(* IEC 61131-3 sources: Bachelor/LARS redcrane-simulation/plc_export/FB_InverceKinematicsVaribleTelescope (part 2) *)

                (* clear; clc; *)
                (* expc3 = [1; 2; 3]; *)
                (* [omghat, theta] = AxisAng3(expc3)   *)

                (* Output: *)
                (* omghat = *)
                (* 0.2673 *)
                (* 0.5345 *)
                (* 0.8018 *)
                (* theta = *)
                (* 3.7417 *)
                (* 'AxisAng3:20' theta = norm(expc3); *)
                (* 'AxisAng3:21' omghat = expc3 / theta; *)
                (* 'MatrixExp6:27' omgmat = se3mat(1: 3, 1: 3) / theta; *)
                FOR i_0 := 0 TO 2 DO
                    omgmat_tmp := DWORD_TO_DINT(SHL(DINT_TO_DWORD(i_0), 2));
                    omgmat[3 * i_0] := se3mat[omgmat_tmp] / c_theta;
                    omgmat[(3 * i_0) + 1] := se3mat[omgmat_tmp + 1] / c_theta;
                    omgmat[(3 * i_0) + 2] := se3mat[omgmat_tmp + 2] / c_theta;
                END_FOR;
                (* 'MatrixExp6:28' T = [MatrixExp3(se3mat(1: 3, 1: 3)), ... *)
                (* 'MatrixExp6:29'          (eye(3) * theta + (1 - cos(theta)) * omgmat ... *)
                (* 'MatrixExp6:30'           + (theta - sin(theta)) * omgmat * omgmat) ... *)
                (* 'MatrixExp6:31'             * se3mat(1: 3, 4) / theta; *)
                (* 'MatrixExp6:32'          0, 0, 0, 1]; *)
                thetalist0_0 := 1.0 - COS(c_theta);
                g_a := c_theta - SIN(c_theta);
                (* *** CHAPTER 3: RIGID-BODY MOTIONS *** *)
                (* Takes a 3x3 so(3) representation of exponential coordinates. *)
                (* Returns R in SO(3) that is achieved by rotating about omghat by theta  *)
                (* from an initial orientation R = I. *)
                (* Example Input: *)

                (* clear; clc; *)
                (* so3mat = [[0, -3, 2]; [3, 0, -1]; [-2, 1, 0]]; *)
                (* R = MatrixExp3(so3mat)   *)

                (* Output: *)
                (* R = *)
                (* -0.6949    0.7135    0.0893 *)
                (* -0.1920   -0.3038    0.9332 *)
                (* 0.6930    0.6313    0.3481 *)
                (* 'MatrixExp3:18' omgtheta = so3ToVec(so3mat); *)
                (* *** CHAPTER 3: RIGID-BODY MOTIONS *** *)
                (* Takes a 3x3 skew-symmetric matrix (an element of so(3)). *)
                (* Returns the corresponding 3-vector (angular velocity). *)
                (* Example Input:  *)

                (* clear; clc; *)
                (* so3mat = [[0, -3, 2]; [3, 0, -1]; [-2, 1, 0]]; *)
                (* omg = so3ToVec(so3mat)   *)

                (* Output: *)
                (* omg = *)
                (* 1 *)
                (* 2 *)
                (* 3 *)
                (* 'so3ToVec:17' omg = [so3mat(3, 2); so3mat(1, 3); so3mat(2, 1)]; *)
                qs4[0] := V[0];
                qs4[1] := V[1];
                qs4[2] := V[2];
                (* 'MatrixExp3:19' if NearZero(norm(omgtheta)) *)
                (* *** BASIC HELPER FUNCTIONS *** *)
                (* Takes a scalar. *)
                (* Checks if the scalar is small enough to be neglected. *)
                (* Example Input: *)

                (* clear; clc; *)
                (* near = -1e-7; *)
                (* judge = NearZero(near) *)

                (* Output: *)
                (* judge = *)
                (* 1 *)
                (* 'NearZero:15' judge = norm(near) < 1e-6; *)
                i_theta := norm(x := qs4);
                IF ABS(i_theta) < 1.0E-6 THEN
                    (* 'MatrixExp3:20' R = eye(3); *)
                    i0_eye();
                    b_R := i0_eye.I;
                ELSE
                    (* 'MatrixExp3:21' else *)
                    (* 'MatrixExp3:22' [omghat, theta] = AxisAng3(omgtheta); *)
                    (* *** CHAPTER 3: RIGID-BODY MOTIONS *** *)
                    (* Takes A 3-vector of exponential coordinates for rotation. *)
                    (* Returns the unit rotation axis omghat and the corresponding rotation  *)
                    (* angle theta. *)
                    (* Example Input: *)

                    (* clear; clc; *)
                    (* expc3 = [1; 2; 3]; *)
                    (* [omghat, theta] = AxisAng3(expc3)   *)

                    (* Output: *)
                    (* omghat = *)
                    (* 0.2673 *)
                    (* 0.5345 *)
                    (* 0.8018 *)
                    (* theta = *)
                    (* 3.7417 *)
                    (* 'AxisAng3:20' theta = norm(expc3); *)
                    (* 'AxisAng3:21' omghat = expc3 / theta; *)
                    (* 'MatrixExp3:23' omgmat = so3mat / theta; *)
                    FOR i_0 := 0 TO 2 DO
                        omgmat_tmp := DWORD_TO_DINT(SHL(DINT_TO_DWORD(i_0), 2));
                        b_omgmat[3 * i_0] := se3mat[omgmat_tmp] / i_theta;
                        b_omgmat[(3 * i_0) + 1] := se3mat[omgmat_tmp + 1] / i_theta;
                        b_omgmat[(3 * i_0) + 2] := se3mat[omgmat_tmp + 2] / i_theta;
                    END_FOR;
                    (* 'MatrixExp3:24' R = eye(3) + sin(theta) * omgmat + (1 - cos(theta)) * omgmat * omgmat; *)
                    l_a := SIN(i_theta);
                    x_tmp := COS(i_theta);
                    i0_eye();
                    tmp := i0_eye.I;
                    FOR i_0 := 0 TO 2 DO
                        FOR omgmat_tmp := 0 TO 2 DO
                            R_tmp := (3 * omgmat_tmp) + i_0;
                            b_R[R_tmp] := (((((1.0 - x_tmp) * b_omgmat[i_0 + 3]) * b_omgmat[(3 * omgmat_tmp) + 1]) + (((1.0 - x_tmp) * b_omgmat[i_0]) * b_omgmat[3 * omgmat_tmp])) + ((b_omgmat[i_0 + 6] * (1.0 - x_tmp)) * b_omgmat[(3 * omgmat_tmp) + 2])) + ((b_omgmat[R_tmp] * l_a) + tmp[R_tmp]);
                        END_FOR;
                    END_FOR;
                END_IF;
                FOR i_0 := 0 TO 2 DO
                    x_tmp := 0.0;
                    FOR omgmat_tmp := 0 TO 2 DO
                        R_tmp := (3 * omgmat_tmp) + i_0;
                        x_tmp := ((((((omgmat[i_0 + 3] * g_a) * omgmat[(3 * omgmat_tmp) + 1]) + ((g_a * omgmat[i_0]) * omgmat[3 * omgmat_tmp])) + ((omgmat[i_0 + 6] * g_a) * omgmat[(3 * omgmat_tmp) + 2])) + ((SINT_TO_LREAL(p_a[R_tmp]) * c_theta) + (omgmat[R_tmp] * thetalist0_0))) * se3mat[omgmat_tmp + 12]) + x_tmp;
                        a[omgmat_tmp + (i_0 * 4)] := b_R[(3 * i_0) + omgmat_tmp];
                    END_FOR;
                    a[i_0 + 12] := x_tmp / c_theta;
                END_FOR;
                a[3] := 0.0;
                a[7] := 0.0;
                a[11] := 0.0;
                a[15] := 1.0;
            END_IF;
            FOR i_0 := 0 TO 3 DO
                thetalist0_0 := T[i_0 + 4];
                g_a := T[i_0];
                l_a := T[i_0 + 8];
                x_tmp := T[i_0 + 12];
                FOR omgmat_tmp := 0 TO 3 DO
                    R_tmp := DWORD_TO_DINT(SHL(DINT_TO_DWORD(omgmat_tmp), 2));
                    M[i_0 + R_tmp] := (((a[R_tmp + 1] * thetalist0_0) + (a[R_tmp] * g_a)) + (a[R_tmp + 2] * l_a)) + (a[R_tmp + 3] * x_tmp);
                END_FOR;
            END_FOR;
            FOR i_0 := 0 TO 15 DO
                T[i_0] := M[i_0];
            END_FOR;
            (* 'JacobianSpace:31' Js(:, i) = Adjoint(T) * Slist(:, i); *)
            (* *** CHAPTER 3: RIGID-BODY MOTIONS *** *)
            (* Takes T a transformation matrix SE3.  *)
            (* Returns the corresponding 6x6 adjoint representation [AdT]. *)
            (* Example Input: *)

            (* clear; clc; *)
            (* T = [[1, 0, 0, 0]; [0, 0, -1, 0]; [0, 1, 0, 3]; [0, 0, 0, 1]]; *)
            (* AdT = Adjoint(T) *)

            (* Output: *)
            (* AdT = *)
            (* 1     0     0     0     0     0 *)
            (* 0     0    -1     0     0     0 *)
            (* 0     1     0     0     0     0 *)
            (* 0     0     3     1     0     0 *)
            (* 3     0     0     0     0    -1 *)
            (* 0     0     0     0     1     0 *)
            (* 'Adjoint:20' [R, p] = TransToRp(T); *)
            (* *** CHAPTER 3: RIGID-BODY MOTIONS *** *)
            (* Takes the transformation matrix T in SE(3)  *)
            (* Returns R: the corresponding rotation matrix *)
            (* p: the corresponding position vector . *)
            (* Example Input: *)

            (* clear; clc; *)
            (* T = [[1, 0, 0, 0]; [0, 0, -1, 0]; [0, 1, 0, 3]; [0, 0, 0, 1]]; *)
            (* [R, p] = TransToRp(T) *)

            (* Output: *)
            (* R = *)
            (* 1     0     0 *)
            (* 0     0    -1 *)
            (* 0     1     0 *)
            (* p = *)
            (* 0 *)
            (* 0 *)
            (* 3 *)
            (* 'TransToRp:22' R = T(1: 3, 1: 3); *)
            (* 'TransToRp:23' p = T(1: 3, 4); *)
            (* 'Adjoint:21' AdT = [R, zeros(3); VecToso3(p) * R, R]; *)
            (* *** CHAPTER 3: RIGID-BODY MOTIONS *** *)
            (* Takes a 3-vector (angular velocity). *)
            (* Returns the skew symmetric matrix in so(3). *)
            (* Example Input: *)

            (* clear; clc; *)
            (* omg = [1; 2; 3]; *)
            (* so3mat = VecToso3(omg) *)

            (* Output: *)
            (* so3mat = *)
            (* 0    -3     2 *)
            (* 3     0    -1 *)
            (* -2     1     0 *)
            (* 'VecToso3:17' so3mat = [0, -omg(3), omg(2); omg(3), 0, -omg(1); -omg(2), omg(1), 0]; *)
            tmp_0[3] :=  -T[14];
            tmp_0[6] := T[13];
            tmp_0[1] := T[14];
            tmp_0[7] :=  -T[12];
            tmp_0[2] :=  -T[13];
            tmp_0[5] := T[12];
            FOR i_0 := 0 TO 2 DO
                x_tmp := tmp_0[i_0 + 3];
                thetalist0_0 := tmp_0[i_0];
                g_a := tmp_0[i_0 + 6];
                FOR omgmat_tmp := 0 TO 2 DO
                    R_tmp := DWORD_TO_DINT(SHL(DINT_TO_DWORD(omgmat_tmp), 2));
                    tmp[i_0 + (3 * omgmat_tmp)] := ((T[R_tmp + 1] * x_tmp) + (T[R_tmp] * thetalist0_0)) + (T[R_tmp + 2] * g_a);
                    Tsb_0[omgmat_tmp + (6 * i_0)] := T[(i_0 * 4) + omgmat_tmp];
                    Tsb_0[omgmat_tmp + (6 * (i_0 + 3))] := 0.0;
                END_FOR;
            END_FOR;
            FOR i_0 := 0 TO 2 DO
                Tsb_0[(6 * i_0) + 3] := tmp[3 * i_0];
                R_tmp := DWORD_TO_DINT(SHL(DINT_TO_DWORD(i_0), 2));
                omgmat_tmp := 6 * (i_0 + 3);
                Tsb_0[omgmat_tmp + 3] := T[R_tmp];
                Tsb_0[(6 * i_0) + 4] := tmp[(3 * i_0) + 1];
                Tsb_0[omgmat_tmp + 4] := T[R_tmp + 1];
                Tsb_0[(6 * i_0) + 5] := tmp[(3 * i_0) + 2];
                Tsb_0[omgmat_tmp + 5] := T[R_tmp + 2];
            END_FOR;
            FOR i_0 := 0 TO 5 DO
                thetalist0_0 := 0.0;
                FOR omgmat_tmp := 0 TO 5 DO
                    thetalist0_0 := (SList[((b_i + 1) * 6) + omgmat_tmp] * Tsb_0[(6 * omgmat_tmp) + i_0]) + thetalist0_0;
                END_FOR;
                Js[i_0 + (6 * (b_i + 1))] := thetalist0_0;
            END_FOR;
        END_FOR;
        (* '<S2>:1:72' Js_pinv = pinv(Js); *)
        (* '<S2>:1:73' xyzDot = [0; *)
        (* '<S2>:1:74'          0; *)
        (* '<S2>:1:75'          0; *)
        (* '<S2>:1:76'          xDot; *)
        (* '<S2>:1:77'          yDot; *)
        (* '<S2>:1:78'          zDot *)
        (* '<S2>:1:79'          ]; *)
        (* '<S2>:1:81' thetaListDot = Js_pinv*xyzDot; *)
        i0_pinv(A := Js);
        tmp_1 := i0_pinv.X;
        (* End of Outputs for SubSystem: '<Root>/FB_InverceKinematicsVaribleTelescope' *)
        (* Outputs for Atomic SubSystem: '<Root>/FB_InverceKinematicsVaribleTelescope' *)
        (* MATLAB Function: '<S1>/inverceKinematics' *)
        V[0] := 0.0;
        V[1] := 0.0;
        V[2] := 0.0;
        V[3] := fXDotRef;
        V[4] := fYDotRef;
        V[5] := fZDotRef;
        (* End of Outputs for SubSystem: '<Root>/FB_InverceKinematicsVaribleTelescope' *)
        (* Outputs for Atomic SubSystem: '<Root>/FB_InverceKinematicsVaribleTelescope' *)
        (* MATLAB Function: '<S1>/inverceKinematics' *)
        FOR i_0 := 0 TO 4 DO
            x_tmp := 0.0;
            FOR omgmat_tmp := 0 TO 5 DO
                x_tmp := (tmp_1[(5 * omgmat_tmp) + i_0] * V[omgmat_tmp]) + x_tmp;
            END_FOR;
            rtb_thetaListDot[i_0] := x_tmp;
        END_FOR;
        (* Update for Memory: '<S1>/Memory' *)
        Memory_PreviousInput[0] := thetalist0[3];
        Memory_PreviousInput[1] := thetalist0[4];
        (* Update for Memory: '<S1>/Memory1' *)
        Memory1_PreviousInput := fKnuckleFeedback;
        (* Update for Memory: '<S1>/Memory2' *)
        Memory2_PreviousInput := fMainFeedback;
        (* Update for Memory: '<S1>/Memory3' *)
        Memory3_PreviousInput := fSlewFeedback;
        (* End of Outputs for SubSystem: '<Root>/FB_InverceKinematicsVaribleTelescope' *)

        (* Outport: '<Root>/fSlewRef' *)
        fSlewRef := thetalist0[0];
        (* Outport: '<Root>/fMainRef' *)
        fMainRef := thetalist0[1];
        (* Outport: '<Root>/fKnuckleRef' *)
        fKnuckleRef := thetalist0[2];
        (* Outport: '<Root>/fSlewVelRef' *)
        fSlewVelRef := rtb_thetaListDot[0];
        (* Outport: '<Root>/fMainVelRef' *)
        fMainVelRef := rtb_thetaListDot[1];
        (* Outport: '<Root>/fKnuckleVelRef' *)
        fKnuckleVelRef := rtb_thetaListDot[2];
        (* Outputs for Atomic SubSystem: '<Root>/FB_InverceKinematicsVaribleTelescope' *)
        (* Outport: '<Root>/success' incorporates:
         *  MATLAB Function: '<S1>/inverceKinematics' *)
        success :=  NOT err;
        (* End of Outputs for SubSystem: '<Root>/FB_InverceKinematicsVaribleTelescope' *)
END_CASE;
END_FUNCTION_BLOCK
FUNCTION isequal: BOOL
VAR_INPUT
    varargin_1: ARRAY [0..8] OF LREAL;
    varargin_2: ARRAY [0..8] OF LREAL;
END_VAR
VAR_TEMP
    b_b_p: BOOL;
    k: DINT;
    exitg1: DINT;
END_VAR
isequal := FALSE;
b_b_p := TRUE;
k := 0;
REPEAT
    exitg1 := 0;
    IF k < 9 THEN
        IF varargin_1[k] <> varargin_2[k] THEN
            b_b_p := FALSE;
            exitg1 := 1;
        ELSE
            k := k + 1;
        END_IF;
    ELSE
        exitg1 := 1;
    END_IF;
UNTIL NOT(exitg1 = 0)
END_REPEAT;
IF b_b_p THEN
    isequal := TRUE;
END_IF;
END_FUNCTION
FUNCTION norm: LREAL
VAR_INPUT
    x: ARRAY [0..2] OF LREAL;
END_VAR
VAR_TEMP
    scale: LREAL;
    absxk: LREAL;
    t: LREAL;
END_VAR
scale := 3.3121686421112381E-170;
absxk := ABS(x[0]);
IF absxk > 3.3121686421112381E-170 THEN
    norm := 1.0;
    scale := absxk;
ELSE
    t := absxk / 3.3121686421112381E-170;
    norm := t * t;
END_IF;
absxk := ABS(x[1]);
IF absxk > scale THEN
    t := scale / absxk;
    norm := ((norm * t) * t) + 1.0;
    scale := absxk;
ELSE
    t := absxk / scale;
    norm := (t * t) + norm;
END_IF;
absxk := ABS(x[2]);
IF absxk > scale THEN
    t := scale / absxk;
    norm := ((norm * t) * t) + 1.0;
    scale := absxk;
ELSE
    t := absxk / scale;
    norm := (t * t) + norm;
END_IF;
norm := scale * SQRT(norm);
END_FUNCTION
FUNCTION_BLOCK pinv
VAR_INPUT
    A: ARRAY [0..29] OF LREAL;
END_VAR
VAR_OUTPUT
    X: ARRAY [0..29] OF LREAL;
END_VAR
VAR
    i0_svd: svd;
END_VAR
VAR_TEMP
    V: ARRAY [0..24] OF LREAL;
    b_r: DINT;
    vcol: DINT;
    U: ARRAY [0..29] OF LREAL;
    b_s: ARRAY [0..4] OF LREAL;
    j: DINT;
    absx: LREAL;
    ia: DINT;
    b: DINT;
    ib: DINT;
    b_ic: DINT;
    ln2x: LREAL;
    e: DINT;
    exitg1: DINT;
    temp2: LREAL;
END_VAR
b_r := -1;
FOR vcol := 0 TO 29 DO
    X[vcol] := 0.0;
END_FOR;
i0_svd(A := A);
U := i0_svd.U;
b_s := i0_svd.b_s;
V := i0_svd.V;
absx := ABS(b_s[0]);
IF absx < 2.2250738585072014E-307 THEN
    ln2x := 2.2250738585072014E-307;
ELSE
    temp2 := LN(absx);
    ln2x := rt_floord(u := temp2 / 0.69314718055994529);
    vcol := TRUNC(ln2x) - 1;
    e :=  -TRUNC(ln2x);
    IF ( -TRUNC(ln2x)) < -1022 THEN
        absx := absx * 1.90109156629516E-211;
        e := 700 - TRUNC(ln2x);
        IF (700 - TRUNC(ln2x)) < -1022 THEN
            absx := absx * 1.90109156629516E-211;
            e := 1400 - TRUNC(ln2x);
        END_IF;
    ELSIF ( -TRUNC(ln2x)) > 1023 THEN
        absx := absx * 5.2601359015483735E+210;
        e := ( -TRUNC(ln2x)) - 700;
        IF (( -TRUNC(ln2x)) - 700) > 1023 THEN
            absx := absx * 5.2601359015483735E+210;
            e := ( -TRUNC(ln2x)) - 1400;
        END_IF;
    END_IF;
    absx := absx * EXPT(2.0, DINT_TO_LREAL(e));
    IF absx < 0.5 THEN
        vcol := TRUNC(ln2x) - 2;
    ELSIF absx >= 1.0 THEN
        vcol := TRUNC(ln2x);
    END_IF;
    ln2x := rt_ldexp_U1d_U2s32_Yd_s_pw(u0 := 1.0, u1 := vcol - 52);
END_IF;
ln2x := 6.0 * ln2x;
vcol := 0;
REPEAT
    exitg1 := 0;
    IF vcol < 5 THEN
        IF b_s[vcol] <= ln2x THEN
            exitg1 := 1;
        ELSE
            b_r := b_r + 1;
            vcol := vcol + 1;
        END_IF;
    ELSE
        exitg1 := 1;
    END_IF;
UNTIL NOT(exitg1 = 0)
END_REPEAT;
IF (b_r + 1) > 0 THEN
    vcol := 0;
    j := 0;
    WHILE j <= b_r DO
        ln2x := 1.0 / b_s[j];
        e := vcol;
        WHILE (e + 1) <= (vcol + 5) DO
            V[e] := ln2x * V[e];
            e := e + 1;
        END_WHILE;
        vcol := vcol + 5;
        j := j + 1;
    END_WHILE;
    FOR vcol := 0 TO 29 DO
        X[vcol] := 0.0;
    END_FOR;
    vcol := 0;
    FOR j := 0 TO 26 BY 5 DO
        e := j;
        WHILE (e + 1) <= (j + 5) DO
            X[e] := 0.0;
            e := e + 1;
        END_WHILE;
    END_FOR;
    FOR j := 0 TO 26 BY 5 DO
        e := -1;
        vcol := vcol + 1;
        b := (6 * b_r) + vcol;
        ib := vcol;
        WHILE ib <= b DO
            ia := e;
            b_ic := j;
            WHILE (b_ic + 1) <= (j + 5) DO
                ia := ia + 1;
                X[b_ic] := (U[ib - 1] * V[ia]) + X[b_ic];
                b_ic := b_ic + 1;
            END_WHILE;
            e := e + 5;
            ib := ib + 6;
        END_WHILE;
    END_FOR;
END_IF;
END_FUNCTION_BLOCK
FUNCTION_BLOCK svd
VAR_INPUT
    A: ARRAY [0..29] OF LREAL;
END_VAR
VAR_OUTPUT
    U: ARRAY [0..29] OF LREAL;
    b_s: ARRAY [0..4] OF LREAL;
    V: ARRAY [0..24] OF LREAL;
END_VAR
VAR
    i0_xzlascl: xzlascl;
    i0_xscal: xscal;
    i0_xscal_f: xscal_f;
    i0_xaxpy_po: xaxpy_po;
    i0_xaxpy_p: xaxpy_p;
    i0_xaxpy: xaxpy;
    i0_xaxpy_poj: xaxpy_poj;
    i0_xscal_fb: xscal_fb;
    i0_xscal_fbq: xscal_fbq;
    i0_xswap: xswap;
    i0_xswap_k: xswap_k;
    i0_xrotg: xrotg;
    i0_xrot: xrot;
    i0_xrot_l: xrot_l;
    i0_xzlascl_g: xzlascl_g;
END_VAR
VAR_TEMP
    b_A: ARRAY [0..29] OF LREAL;
    b_b_s: ARRAY [0..4] OF LREAL;
    e: ARRAY [0..4] OF LREAL;
    work: ARRAY [0..5] OF LREAL;
    Vf: ARRAY [0..24] OF LREAL;
    doscale: BOOL;
    cscale: LREAL;
    anrm: LREAL;
    qq: DINT;
    apply_transform: BOOL;
    nrm: LREAL;
    qjj: DINT;
    qp1jj: DINT;
    m: DINT;
    qp1q: DINT;
    rt: LREAL;
    ztest: LREAL;
    smm1: LREAL;
    emm1: LREAL;
    sqds: LREAL;
    shift: LREAL;
    j_ii: DINT;
    exitg1: DINT;
    temp3: LREAL;
    temp4: LREAL;
    temp5: LREAL;
    temp6: LREAL;
    temp7: LREAL;
    temp8: LREAL;
    temp9: LREAL;
    temp10: LREAL;
    temp11: LREAL;
    temp12: LREAL;
    temp13: LREAL;
    temp14: LREAL;
    temp15: LREAL;
    temp16: LREAL;
END_VAR
FOR m := 0 TO 29 DO
    b_A[m] := A[m];
END_FOR;
FOR m := 0 TO 4 DO
    b_b_s[m] := 0.0;
    e[m] := 0.0;
END_FOR;
FOR m := 0 TO 5 DO
    work[m] := 0.0;
END_FOR;
FOR m := 0 TO 29 DO
    U[m] := 0.0;
END_FOR;
FOR m := 0 TO 24 DO
    Vf[m] := 0.0;
END_FOR;
doscale := FALSE;
anrm := xzlangeM(x := A);
cscale := anrm;
IF (anrm > 0.0) AND (anrm < 6.7178761075670888E-139) THEN
    doscale := TRUE;
    cscale := 6.7178761075670888E-139;
    i0_xzlascl(cfrom := anrm, cto := cscale, m := 6, b_n := 5, A := b_A, iA0 := 1, lda := 6);
ELSIF anrm > 1.4885657073574029E+138 THEN
    doscale := TRUE;
    cscale := 1.4885657073574029E+138;
    i0_xzlascl(cfrom := anrm, cto := cscale, m := 6, b_n := 5, A := b_A, iA0 := 1, lda := 6);
END_IF;
FOR m := 0 TO 4 DO
    qq := (6 * m) + m;
    apply_transform := FALSE;
    nrm := xnrm2(b_n := 6 - m, x := b_A, ix0 := qq + 1);
    IF nrm > 0.0 THEN
        apply_transform := TRUE;
        IF b_A[qq] < 0.0 THEN
            ztest :=  -nrm;
            b_b_s[m] :=  -nrm;
        ELSE
            ztest := nrm;
            b_b_s[m] := nrm;
        END_IF;
        IF ABS(ztest) >= 1.0020841800044864E-292 THEN
            i0_xscal(b_n := 6 - m, a := 1.0 / ztest, x := b_A, ix0 := qq + 1);
        ELSE
            qp1q := (qq - m) + 6;
            qjj := qq;
            WHILE (qjj + 1) <= qp1q DO
                b_A[qjj] := b_A[qjj] / b_b_s[m];
                qjj := qjj + 1;
            END_WHILE;
        END_IF;
        b_A[qq] := b_A[qq] + 1.0;
        b_b_s[m] :=  -b_b_s[m];
    ELSE
        b_b_s[m] := 0.0;
    END_IF;
    qp1q := m + 1;
    WHILE (qp1q + 1) < 6 DO
        qjj := (6 * qp1q) + m;
        IF apply_transform THEN
            temp3 := xdotc(b_n := 6 - m, x := b_A, ix0 := qq + 1, y := b_A, iy0 := qjj + 1);
            i0_xaxpy(b_n := 6 - m, a :=  -(temp3 / b_A[m + (6 * m)]), ix0 := qq + 1, y := b_A, iy0 := qjj + 1);
        END_IF;
        e[qp1q] := b_A[qjj];
        qp1q := qp1q + 1;
    END_WHILE;
    qq := m;
    WHILE (qq + 1) < 7 DO
        U[qq + (6 * m)] := b_A[(6 * m) + qq];
        qq := qq + 1;
    END_WHILE;
    IF (m + 1) <= 3 THEN
        nrm := xnrm2_j(b_n := 4 - m, x := e, ix0 := m + 2);
        IF nrm = 0.0 THEN
            e[m] := 0.0;
        ELSE
            IF e[m + 1] < 0.0 THEN
                e[m] :=  -nrm;
            ELSE
                e[m] := nrm;
            END_IF;
            nrm := e[m];
            IF ABS(e[m]) >= 1.0020841800044864E-292 THEN
                i0_xscal_f(b_n := 4 - m, a := 1.0 / e[m], x := e, ix0 := m + 2);
            ELSE
                qq := m + 1;
                WHILE (qq + 1) <= 5 DO
                    e[qq] := e[qq] / nrm;
                    qq := qq + 1;
                END_WHILE;
            END_IF;
            e[m + 1] := e[m + 1] + 1.0;
            e[m] :=  -e[m];
            qq := m + 1;
            WHILE (qq + 1) < 7 DO
                work[qq] := 0.0;
                qq := qq + 1;
            END_WHILE;
            qq := m + 1;
            WHILE (qq + 1) < 6 DO
                i0_xaxpy_p(b_n := 5 - m, a := e[qq], x := b_A, ix0 := (m + (6 * qq)) + 2, y := work, iy0 := m + 2);
                qq := qq + 1;
            END_WHILE;
            qq := m + 1;
            WHILE (qq + 1) < 6 DO
                i0_xaxpy_po(b_n := 5 - m, a := ( -e[qq]) / e[m + 1], x := work, ix0 := m + 2, y := b_A, iy0 := (m + (6 * qq)) + 2);
                qq := qq + 1;
            END_WHILE;
        END_IF;
        qq := m + 1;
        WHILE (qq + 1) < 6 DO
            Vf[qq + (5 * m)] := e[qq];
            qq := qq + 1;
        END_WHILE;
    END_IF;
END_FOR;
m := 3;
e[3] := b_A[27];
e[4] := 0.0;
FOR qp1q := 4 TO 0 BY -1 DO
    qq := (6 * qp1q) + qp1q;
    IF b_b_s[qp1q] <> 0.0 THEN
        qp1jj := qp1q + 1;
        WHILE (qp1jj + 1) < 6 DO
            qjj := ((6 * qp1jj) + qp1q) + 1;
            temp4 := xdotc(b_n := 6 - qp1q, x := U, ix0 := qq + 1, y := U, iy0 := qjj);
            i0_xaxpy(b_n := 6 - qp1q, a :=  -(temp4 / U[qq]), ix0 := qq + 1, y := U, iy0 := qjj);
            qp1jj := qp1jj + 1;
        END_WHILE;
        qjj := qp1q;
        WHILE (qjj + 1) < 7 DO
            qp1jj := (6 * qp1q) + qjj;
            U[qp1jj] :=  -U[qp1jj];
            qjj := qjj + 1;
        END_WHILE;
        U[qq] := U[qq] + 1.0;
        qq := 0;
        WHILE qq <= (qp1q - 1) DO
            U[qq + (6 * qp1q)] := 0.0;
            qq := qq + 1;
        END_WHILE;
    ELSE
        FOR qjj := 0 TO 5 DO
            U[qjj + (6 * qp1q)] := 0.0;
        END_FOR;
        U[qq] := 1.0;
    END_IF;
END_FOR;
FOR qq := 4 TO 0 BY -1 DO
    IF (qq + 1) <= 3 THEN
        IF e[qq] <> 0.0 THEN
            qp1q := ((5 * qq) + qq) + 2;
            qjj := qq + 1;
            WHILE (qjj + 1) < 6 DO
                qp1jj := ((5 * qjj) + qq) + 2;
                temp5 := xdotc_d(b_n := 4 - qq, x := Vf, ix0 := qp1q, y := Vf, iy0 := qp1jj);
                i0_xaxpy_poj(b_n := 4 - qq, a :=  -(temp5 / Vf[qp1q - 1]), ix0 := qp1q, y := Vf, iy0 := qp1jj);
                qjj := qjj + 1;
            END_WHILE;
        END_IF;
    END_IF;
    FOR qp1q := 0 TO 4 DO
        Vf[qp1q + (5 * qq)] := 0.0;
    END_FOR;
    Vf[qq + (5 * qq)] := 1.0;
END_FOR;
FOR qq := 0 TO 4 DO
    ztest := b_b_s[qq];
    IF ztest <> 0.0 THEN
        rt := ABS(ztest);
        nrm := ztest / rt;
        b_b_s[qq] := rt;
        IF (qq + 1) < 5 THEN
            e[qq] := e[qq] / nrm;
        END_IF;
        i0_xscal_fb(a := nrm, x := U, ix0 := (6 * qq) + 1);
    END_IF;
    IF (qq + 1) < 5 THEN
        nrm := e[qq];
        IF nrm <> 0.0 THEN
            rt := ABS(nrm);
            nrm := rt / nrm;
            e[qq] := rt;
            b_b_s[qq + 1] := b_b_s[qq + 1] * nrm;
            i0_xscal_fbq(a := nrm, x := Vf, ix0 := (5 * (qq + 1)) + 1);
        END_IF;
    END_IF;
END_FOR;
qq := 0;
nrm := 0.0;
FOR qp1q := 0 TO 4 DO
    temp6 := ABS(b_b_s[qp1q]);
    temp7 := ABS(e[qp1q]);
    temp8 := MAX(temp6, temp7);
    nrm := MAX(nrm, temp8);
END_FOR;
WHILE ((m + 2) > 0) AND (qq < 75) DO
    qp1jj := m + 1;
    REPEAT
        exitg1 := 0;
        qp1q := qp1jj;
        IF qp1jj = 0 THEN
            exitg1 := 1;
        ELSE
            rt := ABS(e[qp1jj - 1]);
            IF rt <= ((ABS(b_b_s[qp1jj - 1]) + ABS(b_b_s[qp1jj])) * 2.2204460492503131E-16) THEN
                e[qp1jj - 1] := 0.0;
                exitg1 := 1;
            ELSIF (rt <= 1.0020841800044864E-292) OR ((qq > 20) AND (rt <= (2.2204460492503131E-16 * nrm))) THEN
                e[qp1jj - 1] := 0.0;
                exitg1 := 1;
            ELSE
                qp1jj := qp1jj - 1;
            END_IF;
        END_IF;
    UNTIL NOT(exitg1 = 0)
    END_REPEAT;
    IF (m + 1) = qp1jj THEN
        qp1jj := 4;
    ELSE
        qjj := m + 2;
        j_ii := m + 2;
        REPEAT
            exitg1 := 0;
            IF j_ii >= qp1jj THEN
                qjj := j_ii;
                IF j_ii = qp1jj THEN
                    exitg1 := 1;
                ELSE
                    rt := 0.0;
                    IF j_ii < (m + 2) THEN
                        rt := ABS(e[j_ii - 1]);
                    END_IF;
                    IF j_ii > (qp1jj + 1) THEN
                        rt := ABS(e[j_ii - 2]) + rt;
                    END_IF;
                    ztest := ABS(b_b_s[j_ii - 1]);
                    IF (ztest <= (2.2204460492503131E-16 * rt)) OR (ztest <= 1.0020841800044864E-292) THEN
                        b_b_s[j_ii - 1] := 0.0;
                        exitg1 := 1;
                    ELSE
                        j_ii := j_ii - 1;
                    END_IF;
                END_IF;
            ELSE
                exitg1 := 1;
            END_IF;
        UNTIL NOT(exitg1 = 0)
        END_REPEAT;
        IF qjj = qp1jj THEN
            qp1jj := 3;
        ELSIF (m + 2) = qjj THEN
            qp1jj := 1;
        ELSE
            qp1jj := 2;
            qp1q := qjj;
        END_IF;
    END_IF;
    CASE qp1jj OF
        1:
            rt := e[m];
            e[m] := 0.0;
            qjj := m;
            WHILE (qjj + 1) >= (qp1q + 1) DO
                i0_xrotg(a := b_b_s[qjj], b := rt);
                ztest := i0_xrotg.c;
                sqds := i0_xrotg.b_s;
                IF (qjj + 1) > (qp1q + 1) THEN
                    emm1 := e[qjj - 1];
                    rt := emm1 * ( -sqds);
                    e[qjj - 1] := emm1 * ztest;
                END_IF;
                i0_xrot(x := Vf, ix0 := (5 * qjj) + 1, iy0 := (5 * (m + 1)) + 1, c := ztest, b_s := sqds);
                qjj := qjj - 1;
            END_WHILE;
        2:
            rt := e[qp1q - 1];
            e[qp1q - 1] := 0.0;
            qjj := qp1q;
            WHILE (qjj + 1) <= (m + 2) DO
                i0_xrotg(a := b_b_s[qjj], b := rt);
                ztest := i0_xrotg.c;
                sqds := i0_xrotg.b_s;
                rt := ( -sqds) * e[qjj];
                e[qjj] := e[qjj] * ztest;
                i0_xrot_l(x := U, ix0 := (6 * qjj) + 1, iy0 := (6 * (qp1q - 1)) + 1, c := ztest, b_s := sqds);
                qjj := qjj + 1;
            END_WHILE;
        3:
            rt := b_b_s[m + 1];
            temp9 := ABS(rt);
            temp10 := ABS(b_b_s[m]);
            temp11 := MAX(temp9, temp10);
            temp12 := ABS(e[m]);
            temp13 := MAX(temp11, temp12);
            temp14 := ABS(b_b_s[qp1q]);
            temp15 := MAX(temp13, temp14);
            temp16 := ABS(e[qp1q]);
            ztest := MAX(temp15, temp16);
            rt := rt / ztest;
            smm1 := b_b_s[m] / ztest;
            emm1 := e[m] / ztest;
            sqds := b_b_s[qp1q] / ztest;
            smm1 := (((smm1 + rt) * (smm1 - rt)) + (emm1 * emm1)) / 2.0;
            emm1 := rt * emm1;
            emm1 := emm1 * emm1;
            IF (smm1 <> 0.0) OR (emm1 <> 0.0) THEN
                shift := SQRT((smm1 * smm1) + emm1);
                IF smm1 < 0.0 THEN
                    shift :=  -shift;
                END_IF;
                shift := emm1 / (smm1 + shift);
            ELSE
                shift := 0.0;
            END_IF;
            rt := ((sqds + rt) * (sqds - rt)) + shift;
            ztest := (e[qp1q] / ztest) * sqds;
            qjj := qp1q + 1;
            WHILE qjj <= (m + 1) DO
                i0_xrotg(a := rt, b := ztest);
                sqds := i0_xrotg.c;
                smm1 := i0_xrotg.b_s;
                IF qjj > (qp1q + 1) THEN
                    e[qjj - 2] := rt;
                END_IF;
                emm1 := e[qjj - 1];
                rt := b_b_s[qjj - 1];
                e[qjj - 1] := (emm1 * sqds) - (rt * smm1);
                ztest := smm1 * b_b_s[qjj];
                b_b_s[qjj] := b_b_s[qjj] * sqds;
                i0_xrot(x := Vf, ix0 := (5 * (qjj - 1)) + 1, iy0 := (5 * qjj) + 1, c := sqds, b_s := smm1);
                b_b_s[qjj - 1] := (rt * sqds) + (emm1 * smm1);
                i0_xrotg(a := b_b_s[qjj - 1], b := ztest);
                sqds := i0_xrotg.c;
                smm1 := i0_xrotg.b_s;
                rt := (e[qjj - 1] * sqds) + (smm1 * b_b_s[qjj]);
                b_b_s[qjj] := (e[qjj - 1] * ( -smm1)) + (sqds * b_b_s[qjj]);
                ztest := smm1 * e[qjj];
                e[qjj] := e[qjj] * sqds;
                i0_xrot_l(x := U, ix0 := (6 * (qjj - 1)) + 1, iy0 := (6 * qjj) + 1, c := sqds, b_s := smm1);
                qjj := qjj + 1;
            END_WHILE;
            e[m] := rt;
            qq := qq + 1;
        ELSE
            IF b_b_s[qp1q] < 0.0 THEN
                b_b_s[qp1q] :=  -b_b_s[qp1q];
                i0_xscal_fbq(a := -1.0, x := Vf, ix0 := (5 * qp1q) + 1);
            END_IF;
            qq := qp1q + 1;
            REPEAT
                exitg1 := 0;
                IF (qp1q + 1) < 5 THEN
                    IF b_b_s[qp1q] < b_b_s[qq] THEN
                        rt := b_b_s[qp1q];
                        b_b_s[qp1q] := b_b_s[qq];
                        b_b_s[qq] := rt;
                        i0_xswap(x := Vf, ix0 := (5 * qp1q) + 1, iy0 := (5 * (qp1q + 1)) + 1);
                        i0_xswap_k(x := U, ix0 := (6 * qp1q) + 1, iy0 := (6 * (qp1q + 1)) + 1);
                        qp1q := qq;
                        qq := qq + 1;
                    ELSE
                        exitg1 := 1;
                    END_IF;
                ELSE
                    exitg1 := 1;
                END_IF;
            UNTIL NOT(exitg1 = 0)
            END_REPEAT;
            qq := 0;
            m := m - 1;
    END_CASE;
END_WHILE;
FOR m := 0 TO 4 DO
    b_s[m] := b_b_s[m];
END_FOR;
IF doscale THEN
    i0_xzlascl_g(cfrom := cscale, cto := anrm, m := 5, b_n := 1, A := b_s, iA0 := 1, lda := 5);
END_IF;
FOR m := 0 TO 24 DO
    V[m] := Vf[m];
END_FOR;
END_FUNCTION_BLOCK
FUNCTION xzlangeM: LREAL
VAR_INPUT
    x: ARRAY [0..29] OF LREAL;
END_VAR
VAR_TEMP
    absxk: LREAL;
    k: DINT;
END_VAR
xzlangeM := 0.0;
FOR k := 0 TO 29 DO
    absxk := ABS(x[k]);
    IF absxk > xzlangeM THEN
        xzlangeM := absxk;
    END_IF;
END_FOR;
END_FUNCTION
FUNCTION xnrm2: LREAL
VAR_INPUT
    b_n: DINT;
    x: ARRAY [0..29] OF LREAL;
    ix0: DINT;
END_VAR
VAR_TEMP
    scale: LREAL;
    kend: DINT;
    absxk: LREAL;
    t: LREAL;
    k: DINT;
END_VAR
xnrm2 := 0.0;
IF b_n >= 1 THEN
    IF b_n = 1 THEN
        xnrm2 := ABS(x[ix0 - 1]);
    ELSE
        scale := 3.3121686421112381E-170;
        kend := (ix0 + b_n) - 1;
        k := ix0;
        WHILE k <= kend DO
            absxk := ABS(x[k - 1]);
            IF absxk > scale THEN
                t := scale / absxk;
                xnrm2 := ((xnrm2 * t) * t) + 1.0;
                scale := absxk;
            ELSE
                t := absxk / scale;
                xnrm2 := (t * t) + xnrm2;
            END_IF;
            k := k + 1;
        END_WHILE;
        xnrm2 := scale * SQRT(xnrm2);
    END_IF;
END_IF;
END_FUNCTION
FUNCTION xnrm2_j: LREAL
VAR_INPUT
    b_n: DINT;
    x: ARRAY [0..4] OF LREAL;
    ix0: DINT;
END_VAR
VAR_TEMP
    scale: LREAL;
    kend: DINT;
    absxk: LREAL;
    t: LREAL;
    k: DINT;
END_VAR
xnrm2_j := 0.0;
IF b_n >= 1 THEN
    IF b_n = 1 THEN
        xnrm2_j := ABS(x[ix0 - 1]);
    ELSE
        scale := 3.3121686421112381E-170;
        kend := (ix0 + b_n) - 1;
        k := ix0;
        WHILE k <= kend DO
            absxk := ABS(x[k - 1]);
            IF absxk > scale THEN
                t := scale / absxk;
                xnrm2_j := ((xnrm2_j * t) * t) + 1.0;
                scale := absxk;
            ELSE
                t := absxk / scale;
                xnrm2_j := (t * t) + xnrm2_j;
            END_IF;
            k := k + 1;
        END_WHILE;
        xnrm2_j := scale * SQRT(xnrm2_j);
    END_IF;
END_IF;
END_FUNCTION
FUNCTION_BLOCK xscal
VAR_INPUT
    b_n: DINT;
    a: LREAL;
    ix0: DINT;
END_VAR
VAR_IN_OUT
    x: ARRAY [0..29] OF LREAL;
END_VAR
VAR_TEMP
    b: DINT;
    k: DINT;
END_VAR
b := (ix0 + b_n) - 1;
k := ix0;
WHILE k <= b DO
    x[k - 1] := x[k - 1] * a;
    k := k + 1;
END_WHILE;
END_FUNCTION_BLOCK
FUNCTION_BLOCK xscal_f
VAR_INPUT
    b_n: DINT;
    a: LREAL;
    ix0: DINT;
END_VAR
VAR_IN_OUT
    x: ARRAY [0..4] OF LREAL;
END_VAR
VAR_TEMP
    b: DINT;
    k: DINT;
END_VAR
b := (ix0 + b_n) - 1;
k := ix0;
WHILE k <= b DO
    x[k - 1] := x[k - 1] * a;
    k := k + 1;
END_WHILE;
END_FUNCTION_BLOCK
FUNCTION_BLOCK xaxpy_po
VAR_INPUT
    b_n: DINT;
    a: LREAL;
    x: ARRAY [0..5] OF LREAL;
    ix0: DINT;
    iy0: DINT;
END_VAR
VAR_IN_OUT
    y: ARRAY [0..29] OF LREAL;
END_VAR
VAR_TEMP
    ix: DINT;
    iy: DINT;
    k: DINT;
END_VAR
IF (b_n >= 1) AND (a <> 0.0) THEN
    ix := ix0 - 1;
    iy := iy0 - 1;
    k := 0;
    WHILE k <= (b_n - 1) DO
        y[iy] := (a * x[ix]) + y[iy];
        ix := ix + 1;
        iy := iy + 1;
        k := k + 1;
    END_WHILE;
END_IF;
END_FUNCTION_BLOCK
FUNCTION_BLOCK xaxpy_p
VAR_INPUT
    b_n: DINT;
    a: LREAL;
    x: ARRAY [0..29] OF LREAL;
    ix0: DINT;
    iy0: DINT;
END_VAR
VAR_IN_OUT
    y: ARRAY [0..5] OF LREAL;
END_VAR
VAR_TEMP
    ix: DINT;
    iy: DINT;
    k: DINT;
END_VAR
IF (b_n >= 1) AND (a <> 0.0) THEN
    ix := ix0 - 1;
    iy := iy0 - 1;
    k := 0;
    WHILE k <= (b_n - 1) DO
        y[iy] := (a * x[ix]) + y[iy];
        ix := ix + 1;
        iy := iy + 1;
        k := k + 1;
    END_WHILE;
END_IF;
END_FUNCTION_BLOCK
FUNCTION_BLOCK xaxpy
VAR_INPUT
    b_n: DINT;
    a: LREAL;
    ix0: DINT;
    iy0: DINT;
END_VAR
VAR_IN_OUT
    y: ARRAY [0..29] OF LREAL;
END_VAR
VAR_TEMP
    ix: DINT;
    iy: DINT;
    k: DINT;
END_VAR
IF (b_n >= 1) AND (a <> 0.0) THEN
    ix := ix0 - 1;
    iy := iy0 - 1;
    k := 0;
    WHILE k <= (b_n - 1) DO
        y[iy] := (a * y[ix]) + y[iy];
        ix := ix + 1;
        iy := iy + 1;
        k := k + 1;
    END_WHILE;
END_IF;
END_FUNCTION_BLOCK
FUNCTION_BLOCK xaxpy_poj
VAR_INPUT
    b_n: DINT;
    a: LREAL;
    ix0: DINT;
    iy0: DINT;
END_VAR
VAR_IN_OUT
    y: ARRAY [0..24] OF LREAL;
END_VAR
VAR_TEMP
    ix: DINT;
    iy: DINT;
    k: DINT;
END_VAR
IF (b_n >= 1) AND (a <> 0.0) THEN
    ix := ix0 - 1;
    iy := iy0 - 1;
    k := 0;
    WHILE k <= (b_n - 1) DO
        y[iy] := (a * y[ix]) + y[iy];
        ix := ix + 1;
        iy := iy + 1;
        k := k + 1;
    END_WHILE;
END_IF;
END_FUNCTION_BLOCK
FUNCTION_BLOCK xscal_fb
VAR_INPUT
    a: LREAL;
    ix0: DINT;
END_VAR
VAR_IN_OUT
    x: ARRAY [0..29] OF LREAL;
END_VAR
VAR_TEMP
    k: DINT;
END_VAR
k := ix0;
WHILE k <= (ix0 + 5) DO
    x[k - 1] := x[k - 1] * a;
    k := k + 1;
END_WHILE;
END_FUNCTION_BLOCK
FUNCTION_BLOCK xscal_fbq
VAR_INPUT
    a: LREAL;
    ix0: DINT;
END_VAR
VAR_IN_OUT
    x: ARRAY [0..24] OF LREAL;
END_VAR
VAR_TEMP
    k: DINT;
END_VAR
k := ix0;
WHILE k <= (ix0 + 4) DO
    x[k - 1] := x[k - 1] * a;
    k := k + 1;
END_WHILE;
END_FUNCTION_BLOCK
FUNCTION_BLOCK xswap
VAR_INPUT
    ix0: DINT;
    iy0: DINT;
END_VAR
VAR_IN_OUT
    x: ARRAY [0..24] OF LREAL;
END_VAR
VAR_TEMP
    temp: LREAL;
    k: DINT;
    temp_tmp: DINT;
    tmp: DINT;
END_VAR
FOR k := 0 TO 4 DO
    temp_tmp := (ix0 + k) - 1;
    temp := x[temp_tmp];
    tmp := (iy0 + k) - 1;
    x[temp_tmp] := x[tmp];
    x[tmp] := temp;
END_FOR;
END_FUNCTION_BLOCK
FUNCTION_BLOCK xswap_k
VAR_INPUT
    ix0: DINT;
    iy0: DINT;
END_VAR
VAR_IN_OUT
    x: ARRAY [0..29] OF LREAL;
END_VAR
VAR_TEMP
    temp: LREAL;
    k: DINT;
    temp_tmp: DINT;
    tmp: DINT;
END_VAR
FOR k := 0 TO 5 DO
    temp_tmp := (ix0 + k) - 1;
    temp := x[temp_tmp];
    tmp := (iy0 + k) - 1;
    x[temp_tmp] := x[tmp];
    x[tmp] := temp;
END_FOR;
END_FUNCTION_BLOCK
FUNCTION_BLOCK xrot
VAR_INPUT
    ix0: DINT;
    iy0: DINT;
    c: LREAL;
    b_s: LREAL;
END_VAR
VAR_IN_OUT
    x: ARRAY [0..24] OF LREAL;
END_VAR
VAR_TEMP
    k: DINT;
    temp_tmp: DINT;
    temp_tmp_0: LREAL;
    temp_tmp_1: DINT;
    temp_tmp_2: LREAL;
END_VAR
FOR k := 0 TO 4 DO
    temp_tmp := (iy0 + k) - 1;
    temp_tmp_0 := x[temp_tmp];
    temp_tmp_1 := (ix0 + k) - 1;
    temp_tmp_2 := x[temp_tmp_1];
    x[temp_tmp] := (temp_tmp_0 * c) - (temp_tmp_2 * b_s);
    x[temp_tmp_1] := (temp_tmp_2 * c) + (temp_tmp_0 * b_s);
END_FOR;
END_FUNCTION_BLOCK
FUNCTION_BLOCK xrotg
VAR_OUTPUT
    c: LREAL;
    b_s: LREAL;
END_VAR
VAR_IN_OUT
    a: LREAL;
    b: LREAL;
END_VAR
VAR_TEMP
    roe: LREAL;
    absa: LREAL;
    absb: LREAL;
    scale: LREAL;
    ads: LREAL;
    bds: LREAL;
END_VAR
roe := b;
absa := ABS(a);
absb := ABS(b);
IF absa > absb THEN
    roe := a;
END_IF;
scale := absa + absb;
IF scale = 0.0 THEN
    b_s := 0.0;
    c := 1.0;
    a := 0.0;
    b := 0.0;
ELSE
    ads := absa / scale;
    bds := absb / scale;
    scale := SQRT((ads * ads) + (bds * bds)) * scale;
    IF roe < 0.0 THEN
        scale :=  -scale;
    END_IF;
    c := a / scale;
    b_s := b / scale;
    IF absa > absb THEN
        b := b_s;
    ELSIF c <> 0.0 THEN
        b := 1.0 / c;
    ELSE
        b := 1.0;
    END_IF;
    a := scale;
END_IF;
END_FUNCTION_BLOCK
FUNCTION_BLOCK xrot_l
VAR_INPUT
    ix0: DINT;
    iy0: DINT;
    c: LREAL;
    b_s: LREAL;
END_VAR
VAR_IN_OUT
    x: ARRAY [0..29] OF LREAL;
END_VAR
VAR_TEMP
    k: DINT;
    temp_tmp: DINT;
    temp_tmp_0: LREAL;
    temp_tmp_1: DINT;
    temp_tmp_2: LREAL;
END_VAR
FOR k := 0 TO 5 DO
    temp_tmp := (iy0 + k) - 1;
    temp_tmp_0 := x[temp_tmp];
    temp_tmp_1 := (ix0 + k) - 1;
    temp_tmp_2 := x[temp_tmp_1];
    x[temp_tmp] := (temp_tmp_0 * c) - (temp_tmp_2 * b_s);
    x[temp_tmp_1] := (temp_tmp_2 * c) + (temp_tmp_0 * b_s);
END_FOR;
END_FUNCTION_BLOCK
FUNCTION_BLOCK xzlascl_g
VAR_INPUT
    cfrom: LREAL;
    cto: LREAL;
    m: DINT;
    b_n: DINT;
    iA0: DINT;
    lda: DINT;
END_VAR
VAR_IN_OUT
    A: ARRAY [0..4] OF LREAL;
END_VAR
VAR_TEMP
    cfromc: LREAL;
    ctoc: LREAL;
    notdone: BOOL;
    cfrom1: LREAL;
    cto1: LREAL;
    b_mul: LREAL;
    offset: DINT;
    j: DINT;
    i: DINT;
    tmp: DINT;
    temp1: BOOL;
END_VAR
cfromc := cfrom;
ctoc := cto;
notdone := TRUE;
WHILE notdone DO
    cfrom1 := cfromc * 2.0041683600089728E-292;
    cto1 := ctoc / 4.9896007738368E+291;
    temp1 := FALSE;
    IF ABS(cfrom1) > ABS(ctoc) THEN
        IF ctoc <> 0.0 THEN
            b_mul := 2.0041683600089728E-292;
            cfromc := cfrom1;
        ELSE
            temp1 := TRUE;
        END_IF;
    ELSE
        temp1 := TRUE;
    END_IF;
    IF temp1 THEN
        IF ABS(cto1) > ABS(cfromc) THEN
            b_mul := 4.9896007738368E+291;
            ctoc := cto1;
        ELSE
            b_mul := ctoc / cfromc;
            notdone := FALSE;
        END_IF;
    END_IF;
    j := 0;
    WHILE j <= (b_n - 1) DO
        offset := ((j * lda) + iA0) - 2;
        i := 1;
        WHILE (i - 1) <= (m - 1) DO
            tmp := offset + i;
            A[tmp] := A[tmp] * b_mul;
            i := i + 1;
        END_WHILE;
        j := j + 1;
    END_WHILE;
END_WHILE;
END_FUNCTION_BLOCK
FUNCTION_BLOCK xzlascl
VAR_INPUT
    cfrom: LREAL;
    cto: LREAL;
    m: DINT;
    b_n: DINT;
    iA0: DINT;
    lda: DINT;
END_VAR
VAR_IN_OUT
    A: ARRAY [0..29] OF LREAL;
END_VAR
VAR_TEMP
    cfromc: LREAL;
    ctoc: LREAL;
    notdone: BOOL;
    cfrom1: LREAL;
    cto1: LREAL;
    b_mul: LREAL;
    offset: DINT;
    j: DINT;
    i: DINT;
    tmp: DINT;
    temp1: BOOL;
END_VAR
cfromc := cfrom;
ctoc := cto;
notdone := TRUE;
WHILE notdone DO
    cfrom1 := cfromc * 2.0041683600089728E-292;
    cto1 := ctoc / 4.9896007738368E+291;
    temp1 := FALSE;
    IF ABS(cfrom1) > ABS(ctoc) THEN
        IF ctoc <> 0.0 THEN
            b_mul := 2.0041683600089728E-292;
            cfromc := cfrom1;
        ELSE
            temp1 := TRUE;
        END_IF;
    ELSE
        temp1 := TRUE;
    END_IF;
    IF temp1 THEN
        IF ABS(cto1) > ABS(cfromc) THEN
            b_mul := 4.9896007738368E+291;
            ctoc := cto1;
        ELSE
            b_mul := ctoc / cfromc;
            notdone := FALSE;
        END_IF;
    END_IF;
    j := 0;
    WHILE j <= (b_n - 1) DO
        offset := ((j * lda) + iA0) - 2;
        i := 1;
        WHILE (i - 1) <= (m - 1) DO
            tmp := offset + i;
            A[tmp] := A[tmp] * b_mul;
            i := i + 1;
        END_WHILE;
        j := j + 1;
    END_WHILE;
END_WHILE;
END_FUNCTION_BLOCK
FUNCTION xdotc: LREAL
VAR_INPUT
    b_n: DINT;
    x: ARRAY [0..29] OF LREAL;
    ix0: DINT;
    y: ARRAY [0..29] OF LREAL;
    iy0: DINT;
END_VAR
VAR_TEMP
    ix: DINT;
    iy: DINT;
    k: DINT;
END_VAR
xdotc := 0.0;
IF b_n >= 1 THEN
    ix := ix0;
    iy := iy0;
    k := 0;
    WHILE k <= (b_n - 1) DO
        xdotc := (x[ix - 1] * y[iy - 1]) + xdotc;
        ix := ix + 1;
        iy := iy + 1;
        k := k + 1;
    END_WHILE;
END_IF;
END_FUNCTION
FUNCTION xdotc_d: LREAL
VAR_INPUT
    b_n: DINT;
    x: ARRAY [0..24] OF LREAL;
    ix0: DINT;
    y: ARRAY [0..24] OF LREAL;
    iy0: DINT;
END_VAR
VAR_TEMP
    ix: DINT;
    iy: DINT;
    k: DINT;
END_VAR
xdotc_d := 0.0;
IF b_n >= 1 THEN
    ix := ix0;
    iy := iy0;
    k := 0;
    WHILE k <= (b_n - 1) DO
        xdotc_d := (x[ix - 1] * y[iy - 1]) + xdotc_d;
        ix := ix + 1;
        iy := iy + 1;
        k := k + 1;
    END_WHILE;
END_IF;
END_FUNCTION
FUNCTION rt_floord: LREAL
VAR_INPUT
    u: LREAL;
END_VAR
rt_floord := DINT_TO_LREAL(TRUNC(u));
IF u = rt_floord THEN
    rt_floord := u;
ELSIF u < 0.0 THEN
    rt_floord := rt_floord - 1.0;
END_IF;
END_FUNCTION
FUNCTION rt_ldexp_U1d_U2s32_Yd_s_pw: LREAL
VAR_INPUT
    u0: LREAL;
    u1: DINT;
END_VAR
IF (u0 = 0.0) OR (u1 = 0) THEN
    rt_ldexp_U1d_U2s32_Yd_s_pw := u0;
ELSE
    rt_ldexp_U1d_U2s32_Yd_s_pw := u0 * EXPT(2.0, DINT_TO_LREAL(u1));
END_IF;
END_FUNCTION
FUNCTION_BLOCK eye
VAR_OUTPUT
    I: ARRAY [0..8] OF LREAL;
END_VAR
VAR_TEMP
    b_i: DINT;
END_VAR
FOR b_i := 0 TO 8 DO
    I[b_i] := 0.0;
END_FOR;
I[0] := 1.0;
I[4] := 1.0;
I[8] := 1.0;
END_FUNCTION_BLOCK
FUNCTION_BLOCK MatrixLog3
VAR_INPUT
    b_R: ARRAY [0..8] OF LREAL;
END_VAR
VAR_OUTPUT
    so3mat: ARRAY [0..8] OF LREAL;
END_VAR
VAR_TEMP
    acosinput: LREAL;
    theta: LREAL;
    t: LREAL;
    i: DINT;
    b_idx_0: LREAL;
    b_idx_1: LREAL;
    so3mat_tmp: DINT;
END_VAR
(* 'MatrixLog3:18' acosinput = (trace(R) - 1) / 2; *)
acosinput := (((b_R[0] + b_R[4]) + b_R[8]) - 1.0) / 2.0;
(* 'MatrixLog3:19' if acosinput >= 1 *)
IF acosinput >= 1.0 THEN
    (* 'MatrixLog3:20' so3mat = zeros(3); *)
    FOR i := 0 TO 8 DO
        so3mat[i] := 0.0;
    END_FOR;
ELSIF acosinput <= -1.0 THEN
    (* 'MatrixLog3:21' elseif acosinput <= -1 *)
    (* 'MatrixLog3:22' if ~NearZero(1 + R(3, 3)) *)
    (* *** BASIC HELPER FUNCTIONS *** *)
    (* Takes a scalar. *)
    (* Checks if the scalar is small enough to be neglected. *)
    (* Example Input: *)

    (* clear; clc; *)
    (* near = -1e-7; *)
    (* judge = NearZero(near) *)

    (* Output: *)
    (* judge = *)
    (* 1 *)
    (* 'NearZero:15' judge = norm(near) < 1e-6; *)
    IF ABS(b_R[8] + 1.0) >= 1.0E-6 THEN
        (* 'MatrixLog3:23' omg = (1 / sqrt(2 * (1 + R(3, 3)))) ... *)
        (* 'MatrixLog3:24'               * [R(1, 3); R(2, 3); 1 + R(3, 3)]; *)
        t := 1.0 / SQRT((b_R[8] + 1.0) * 2.0);
        b_idx_0 := t * b_R[6];
        b_idx_1 := t * b_R[7];
        t := (b_R[8] + 1.0) * t;
    ELSE
        (* *** BASIC HELPER FUNCTIONS *** *)
        (* Takes a scalar. *)
        (* Checks if the scalar is small enough to be neglected. *)
        (* Example Input: *)

        (* clear; clc; *)
        (* near = -1e-7; *)
        (* judge = NearZero(near) *)

        (* Output: *)
        (* judge = *)
        (* 1 *)
        (* 'NearZero:15' judge = norm(near) < 1e-6; *)
        IF ABS(b_R[4] + 1.0) >= 1.0E-6 THEN
            (* 'MatrixLog3:25' elseif ~NearZero(1 + R(2, 2)) *)
            (* 'MatrixLog3:26' omg = (1 / sqrt(2 * (1 + R(2, 2)))) ... *)
            (* 'MatrixLog3:27'               * [R(1, 2); 1 + R(2, 2); R(3, 2)]; *)
            t := 1.0 / SQRT((b_R[4] + 1.0) * 2.0);
            b_idx_0 := t * b_R[3];
            b_idx_1 := (b_R[4] + 1.0) * t;
            t := t * b_R[5];
        ELSE
            (* 'MatrixLog3:28' else *)
            (* 'MatrixLog3:29' omg = (1 / sqrt(2 * (1 + R(1, 1)))) ... *)
            (* 'MatrixLog3:30'               * [1 + R(1, 1); R(2, 1); R(3, 1)]; *)
            t := 1.0 / SQRT((b_R[0] + 1.0) * 2.0);
            b_idx_0 := (b_R[0] + 1.0) * t;
            b_idx_1 := t * b_R[1];
            t := t * b_R[2];
        END_IF;
    END_IF;
    (* 'MatrixLog3:32' so3mat = VecToso3(pi * omg); *)
    b_idx_0 := 3.1415926535897931 * b_idx_0;
    b_idx_1 := 3.1415926535897931 * b_idx_1;
    t := 3.1415926535897931 * t;
    (* *** CHAPTER 3: RIGID-BODY MOTIONS *** *)
    (* Takes a 3-vector (angular velocity). *)
    (* Returns the skew symmetric matrix in so(3). *)
    (* Example Input: *)

    (* clear; clc; *)
    (* omg = [1; 2; 3]; *)
    (* so3mat = VecToso3(omg) *)

    (* Output: *)
    (* so3mat = *)
    (* 0    -3     2 *)
    (* 3     0    -1 *)
    (* -2     1     0 *)
    (* 'VecToso3:17' so3mat = [0, -omg(3), omg(2); omg(3), 0, -omg(1); -omg(2), omg(1), 0]; *)
    so3mat[0] := 0.0;
    so3mat[3] :=  -t;
    so3mat[6] := b_idx_1;
    so3mat[1] := t;
    so3mat[4] := 0.0;
    so3mat[7] :=  -b_idx_0;
    so3mat[2] :=  -b_idx_1;
    so3mat[5] := b_idx_0;
    so3mat[8] := 0.0;
ELSE
    (* 'MatrixLog3:33' else *)
    (* 'MatrixLog3:34' theta = acos(acosinput); *)
    theta := ACOS(acosinput);
    (* 'MatrixLog3:35' so3mat = theta * (1 / (2 * sin(theta))) * (R - R'); *)
    t := (1.0 / (2.0 * SIN(theta))) * theta;
    FOR i := 0 TO 2 DO
        so3mat[3 * i] := (b_R[3 * i] - b_R[i]) * t;
        so3mat_tmp := (3 * i) + 1;
        so3mat[so3mat_tmp] := (b_R[so3mat_tmp] - b_R[i + 3]) * t;
        so3mat_tmp := (3 * i) + 2;
        so3mat[so3mat_tmp] := (b_R[so3mat_tmp] - b_R[i + 6]) * t;
    END_FOR;
END_IF;
END_FUNCTION_BLOCK
VAR_GLOBAL CONSTANT
    SS_INITIALIZE: SINT := 0;
    SS_STEP: SINT := 1;
END_VAR
